FUNCTION_BLOCK ST001 EXTENDS TcoCore.TcoObject
VAR	
	{attribute addProperty Name "<#MANUAL#>"}
	_serviceModeTask : TcoCore.TcoTask(THIS^);
    {attribute addProperty Name "<#GROUND#>"}	
	_groundSequenceTask  : TcoCore.TcoTask(THIS^);
	{attribute addProperty Name "<#AUTOMAT#>"}	
	_automatSequenceTask  : TcoCore.TcoTask(THIS^);
	
	{attribute clr [Container(Layout.Stack)]}
	_components : ST001_ComponentsHandler(THIS^);
	
	{attribute clr [RenderIgnore()]}
	_mqttMirrorComponents : ST001_ComponentsHandler(THIS^);
	
	{attribute clr [Container(Layout.Stack)]}
	_groundPositionSequence : ST001_GroundSequence(THIS^, eRestoreMode.None);
	_automatPositionSequence : ST001_AutomatSequence(THIS^, eRestoreMode.None);
	
	_settings 	: ST001_ProcessDataManager(THIS^);
	_repository : ST001_ProcessDataManager(THIS^);
END_VAR

_components();
_settings();
_repository();
_groundPositionSequence(inoComponents := _components);
_automatPositionSequence(inoComponents := _components);


IF(_groundSequenceTask.Execute()) THEN
	_serviceModeTask.Abort();
	_groundPositionSequence.Run();
	_groundSequenceTask.DoneWhen(_groundPositionSequence.CurrentStep.ID = _groundPositionSequence.MaxStepID - 1);	
END_IF

_automatSequenceTask.Enabled := _groundSequenceTask.Done;

IF(_automatSequenceTask.Execute()) THEN	
	_automatPositionSequence.Run();
END_IF

IF(_serviceModeTask.Execute()) THEN
	_automatSequenceTask.Restore();	
	_groundSequenceTask.Restore();
	_groundPositionSequence.Restore();
	_components.Service();
END_IF

PROPERTY Repository : REFERENCE TO ST001_ProcessDataManager
GET
Repository REF= _repository;
END_GET
END_PROPERTY

PROPERTY Settings : REFERENCE TO ST001_ProcessDataManager
GET
Settings REF= _settings;
END_GET
END_PROPERTY

END_FUNCTION_BLOCK

(* stored: Version 1.1.0.1
   POU ST001: Id {010cafc4-622f-0b8f-2fed-ee2ff87a3f00}, SpecialFunc None
   Property Repository: Id {cb48c119-fade-018a-3a85-7fcfa6a3b0dc}
   Get Get: Id {66fbcbe4-e4c7-0b70-37e7-078bc6baa61a}
   Property Settings: Id {4ad2c757-2f00-04a2-2663-bb2411c40db7}
   Get Get: Id {6bdeca15-35a6-090c-2d41-cde43739ad03} *)
